TYPE ST_Intern_Interpreter :
STRUCT
	
		
END_STRUCT
END_TYPE

(* stored: Version 1.1.0.1, ProductVersion 3.1.4019.2
   DUT ST_Intern_Interpreter: Id {96345b14-1396-4321-97ca-2fedd5a41ebb} *)
